(* Logix 5000 project; controller DispersionPlc vendor 1 type 14 code 108 rev 34.11; software revision 34.01; part 22 of 22 *)
(* tags used below, declared in another part *)
   AFI : BOOL;
   DeviationFactor : REAL;
   Estop : BOOL;
   Estop_Disp : ALIAS FOR Local:3:I.Data.1;
   FC_4302_1 : AStd_PIDInterface;
   FC_4302_1_AOI : AStd_PIDInterface_AOI;
   FC_4302_1_PID : PID_ENHANCED;
   FCV_4302_1 : AStd_VlvModulating;
   FIT_4302_2 : AStd_AnalogInput;
   GenPurp : AStd_GeneralPurp;
   LS_4302_High : BOOL;
   PLCStatus : AStd_PLCStatus;
   RO_HE4305_PhaseROWaterAddition : AStd_PLI;
   SV_4307_1 : AStd_VlvOC;
   TIT_4307_1 : AStd_AnalogInput;
   V4306_PhaseTransfer : AStd_PLI;
   V4307_PhaseCool : AStd_PLI;
   V4307_PhaseCool_AOI : AStd_PLI_AOI;
   V4307_PhaseRunPumpCirculate : AStd_PLI;
   V4307_PhaseRunPumpCirculate_AOI : AStd_PLI_AOI;
   V4307_PhaseTransfer : AStd_PLI;
   V4307_PhaseTransfer_AOI : AStd_PLI_AOI;
   V4307_PhaseTransfer_DelayTimer : TIMER;
   V4307_Transfer_LineClear : TIMER;
   VFD_4302_1 : AStd_VFD;
   VFD_4307_1 : AStd_VFD;
   WIT_4307_1 : AStd_AnalogInput;
   XV_4302_10 : AStd_VlvOC;
   XV_4306_5 : AStd_VlvOC;
   XV_4307_1 : AStd_VlvOC;
   XV_4307_2 : AStd_VlvOC;
   XV_4307_4 : AStd_VlvOC;
   XV_4307_6 : AStd_VlvOC;
(* Unit_V4307, continued *)

ROUTINE Phase_Cool   (* ladder *)
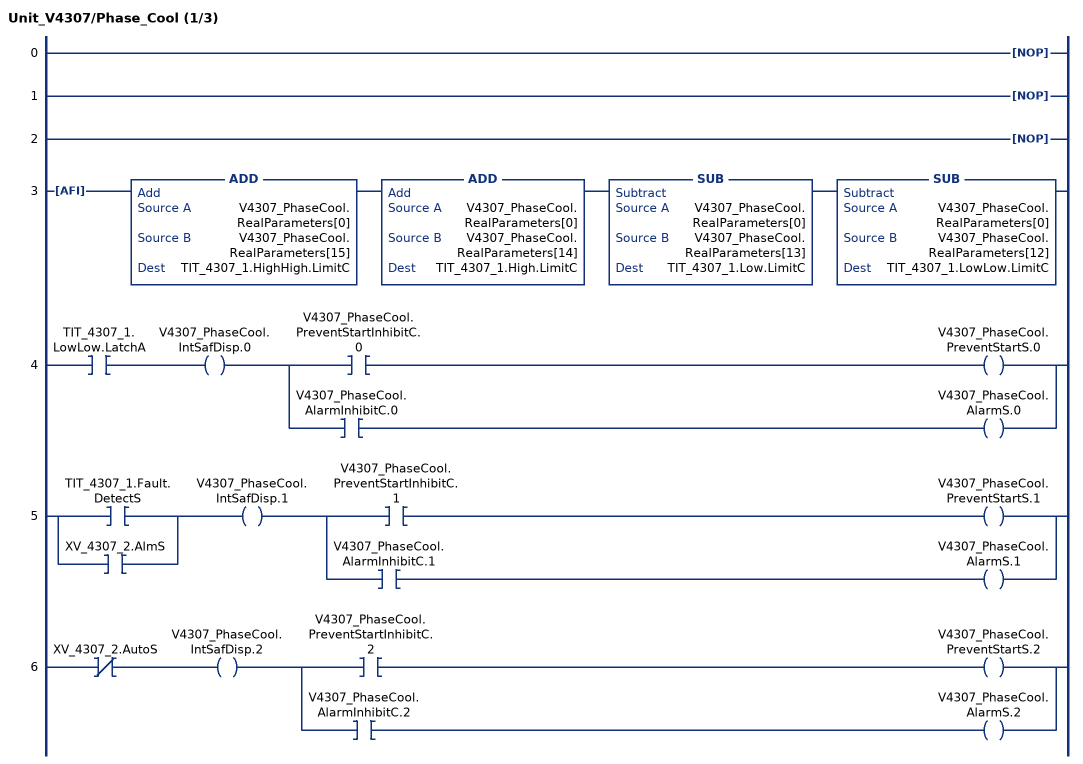
   0: NOP();
   1: NOP();
   2: NOP();
   3: AFI()ADD(V4307_PhaseCool.RealParameters[0],V4307_PhaseCool.RealParameters[15],TIT_4307_1.HighHigh.LimitC)ADD(V4307_PhaseCool.RealParameters[0],V4307_PhaseCool.RealParameters[14],TIT_4307_1.High.LimitC)SUB(V4307_PhaseCool.RealParameters[0],V4307_PhaseCool.RealParameters[13],TIT_4307_1.Low.LimitC)SUB(V4307_PhaseCool.RealParameters[0],V4307_PhaseCool.RealParameters[12],TIT_4307_1.LowLow.LimitC);
   4: XIC(TIT_4307_1.LowLow.LatchA)OTE(V4307_PhaseCool.IntSafDisp.0)[XIC(V4307_PhaseCool.PreventStartInhibitC.0) OTE(V4307_PhaseCool.PreventStartS.0) ,XIC(V4307_PhaseCool.AlarmInhibitC.0) OTE(V4307_PhaseCool.AlarmS.0) ];
   5: [XIC(TIT_4307_1.Fault.DetectS) ,XIC(XV_4307_2.AlmS) ]OTE(V4307_PhaseCool.IntSafDisp.1)[XIC(V4307_PhaseCool.PreventStartInhibitC.1) OTE(V4307_PhaseCool.PreventStartS.1) ,XIC(V4307_PhaseCool.AlarmInhibitC.1) OTE(V4307_PhaseCool.AlarmS.1) ];
   6: XIO(XV_4307_2.AutoS)OTE(V4307_PhaseCool.IntSafDisp.2)[XIC(V4307_PhaseCool.PreventStartInhibitC.2) OTE(V4307_PhaseCool.PreventStartS.2) ,XIC(V4307_PhaseCool.AlarmInhibitC.2) OTE(V4307_PhaseCool.AlarmS.2) ];
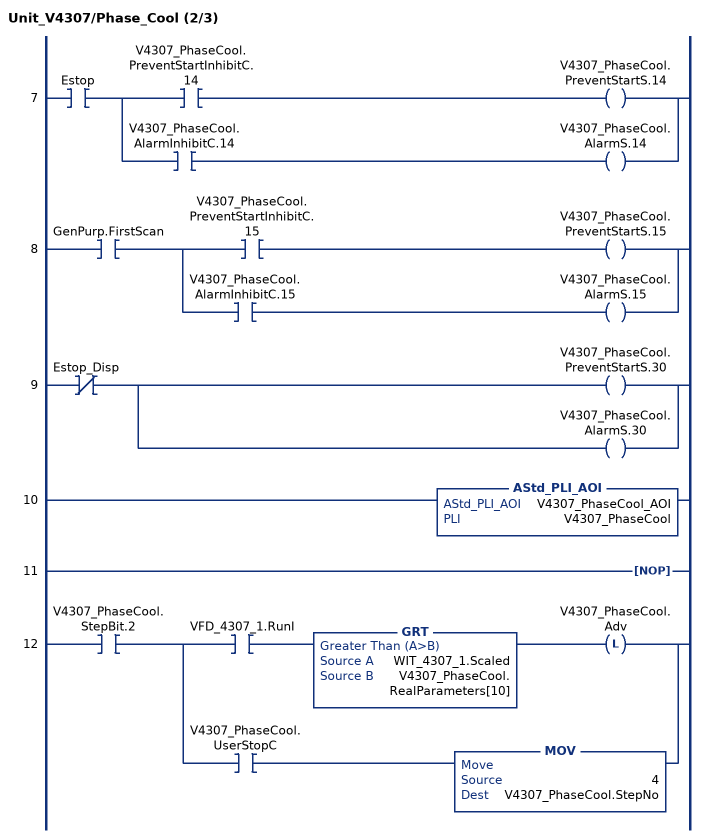
   7: XIC(Estop)[XIC(V4307_PhaseCool.PreventStartInhibitC.14) OTE(V4307_PhaseCool.PreventStartS.14) ,XIC(V4307_PhaseCool.AlarmInhibitC.14) OTE(V4307_PhaseCool.AlarmS.14) ];
   8: XIC(GenPurp.FirstScan)[XIC(V4307_PhaseCool.PreventStartInhibitC.15) OTE(V4307_PhaseCool.PreventStartS.15) ,XIC(V4307_PhaseCool.AlarmInhibitC.15) OTE(V4307_PhaseCool.AlarmS.15) ];
   9: XIO(Estop_Disp)[OTE(V4307_PhaseCool.PreventStartS.30) ,OTE(V4307_PhaseCool.AlarmS.30) ];
   10: AStd_PLI_AOI(V4307_PhaseCool_AOI,V4307_PhaseCool);
   11: NOP();
   12: XIC(V4307_PhaseCool.StepBit.2)[XIC(VFD_4307_1.RunI) GRT(WIT_4307_1.Scaled,V4307_PhaseCool.RealParameters[10]) OTL(V4307_PhaseCool.Adv) ,XIC(V4307_PhaseCool.UserStopC) MOV(4,V4307_PhaseCool.StepNo) ];
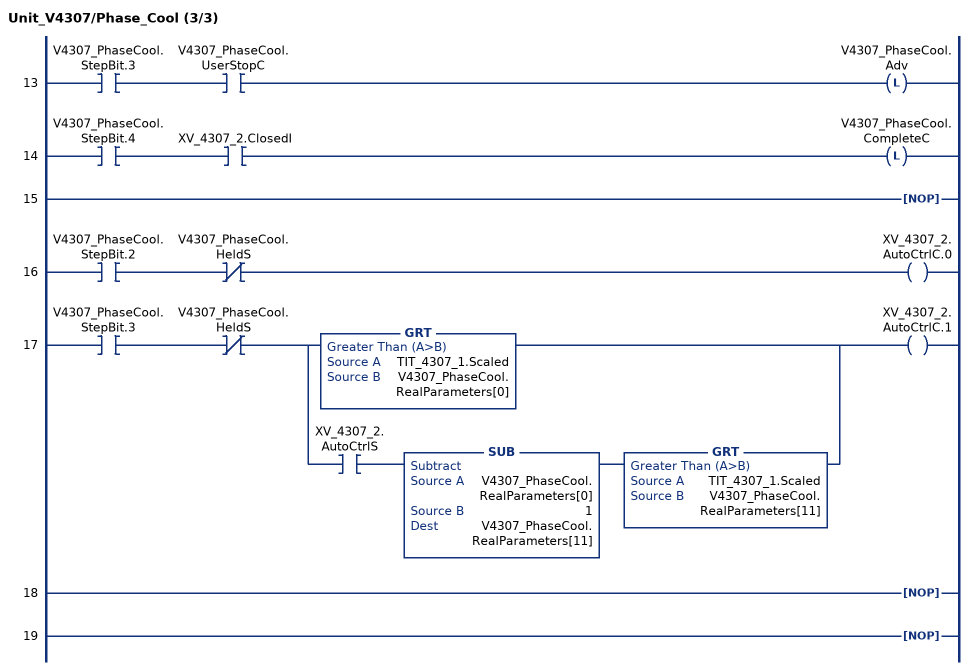
   13: XIC(V4307_PhaseCool.StepBit.3)XIC(V4307_PhaseCool.UserStopC)OTL(V4307_PhaseCool.Adv);
   14: XIC(V4307_PhaseCool.StepBit.4)XIC(XV_4307_2.ClosedI)OTL(V4307_PhaseCool.CompleteC);
   15: NOP();
   16: XIC(V4307_PhaseCool.StepBit.2)XIO(V4307_PhaseCool.HeldS)OTE(XV_4307_2.AutoCtrlC.0);
   17: XIC(V4307_PhaseCool.StepBit.3)XIO(V4307_PhaseCool.HeldS)[GRT(TIT_4307_1.Scaled,V4307_PhaseCool.RealParameters[0]) ,XIC(XV_4307_2.AutoCtrlS) SUB(V4307_PhaseCool.RealParameters[0],1,V4307_PhaseCool.RealParameters[11]) GRT(TIT_4307_1.Scaled,V4307_PhaseCool.RealParameters[11]) ]OTE(XV_4307_2.AutoCtrlC.1);
   18: NOP();
   19: NOP();
END_ROUTINE

ROUTINE Phase_RunPump_Circulate   (* ladder *)
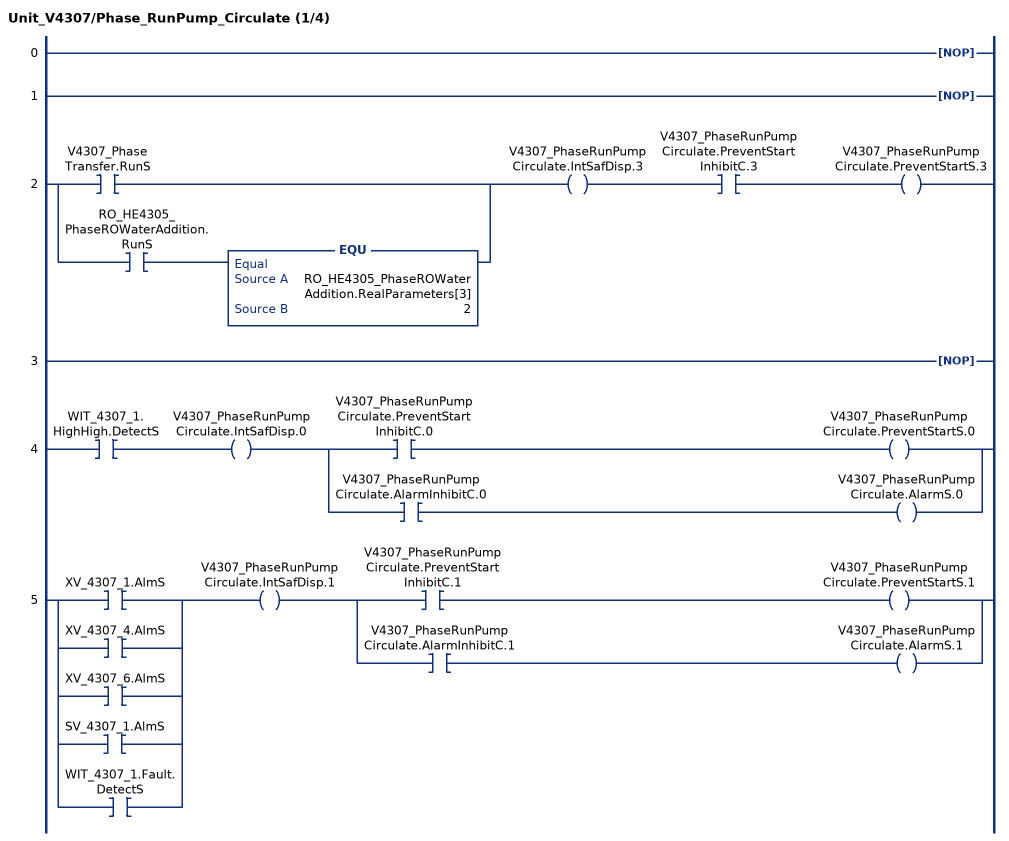
   0: NOP();
   1: NOP();
   2: [XIC(V4307_PhaseTransfer.RunS) ,XIC(RO_HE4305_PhaseROWaterAddition.RunS) EQU(RO_HE4305_PhaseROWaterAddition.RealParameters[3],2) ]OTE(V4307_PhaseRunPumpCirculate.IntSafDisp.3)XIC(V4307_PhaseRunPumpCirculate.PreventStartInhibitC.3)OTE(V4307_PhaseRunPumpCirculate.PreventStartS.3);
   3: NOP();
   4: XIC(WIT_4307_1.HighHigh.DetectS)OTE(V4307_PhaseRunPumpCirculate.IntSafDisp.0)[XIC(V4307_PhaseRunPumpCirculate.PreventStartInhibitC.0) OTE(V4307_PhaseRunPumpCirculate.PreventStartS.0) ,XIC(V4307_PhaseRunPumpCirculate.AlarmInhibitC.0) OTE(V4307_PhaseRunPumpCirculate.AlarmS.0) ];
   5: [XIC(XV_4307_1.AlmS) ,XIC(XV_4307_4.AlmS) ,XIC(XV_4307_6.AlmS) ,XIC(SV_4307_1.AlmS) ,XIC(WIT_4307_1.Fault.DetectS) ]OTE(V4307_PhaseRunPumpCirculate.IntSafDisp.1)[XIC(V4307_PhaseRunPumpCirculate.PreventStartInhibitC.1) OTE(V4307_PhaseRunPumpCirculate.PreventStartS.1) ,XIC(V4307_PhaseRunPumpCirculate.AlarmInhibitC.1) OTE(V4307_PhaseRunPumpCirculate.AlarmS.1) ];
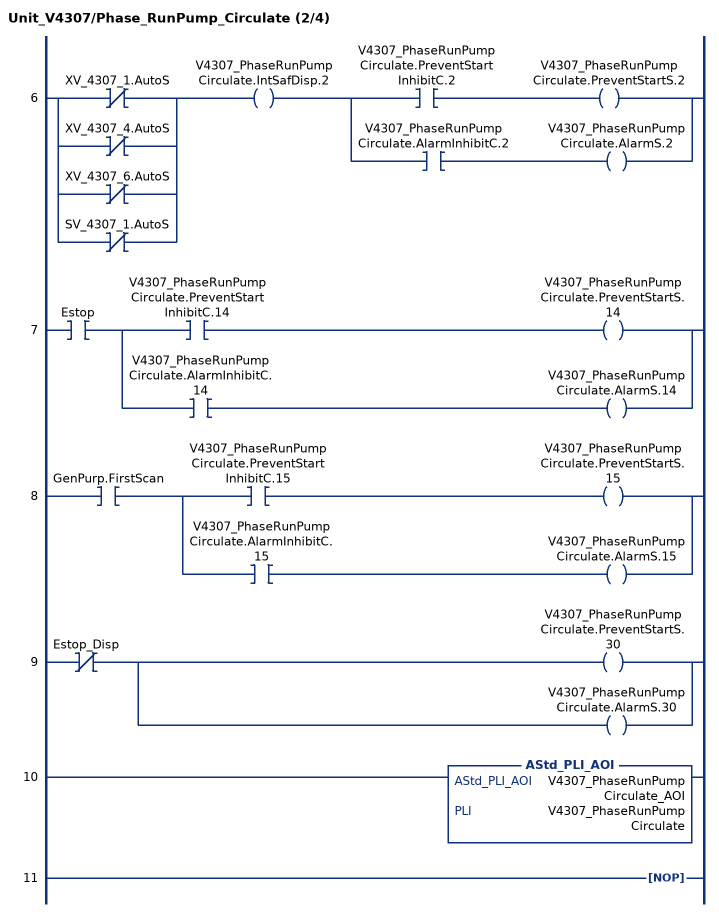
   6: [XIO(XV_4307_1.AutoS) ,XIO(XV_4307_4.AutoS) ,XIO(XV_4307_6.AutoS) ,XIO(SV_4307_1.AutoS) ]OTE(V4307_PhaseRunPumpCirculate.IntSafDisp.2)[XIC(V4307_PhaseRunPumpCirculate.PreventStartInhibitC.2) OTE(V4307_PhaseRunPumpCirculate.PreventStartS.2) ,XIC(V4307_PhaseRunPumpCirculate.AlarmInhibitC.2) OTE(V4307_PhaseRunPumpCirculate.AlarmS.2) ];
   7: XIC(Estop)[XIC(V4307_PhaseRunPumpCirculate.PreventStartInhibitC.14) OTE(V4307_PhaseRunPumpCirculate.PreventStartS.14) ,XIC(V4307_PhaseRunPumpCirculate.AlarmInhibitC.14) OTE(V4307_PhaseRunPumpCirculate.AlarmS.14) ];
   8: XIC(GenPurp.FirstScan)[XIC(V4307_PhaseRunPumpCirculate.PreventStartInhibitC.15) OTE(V4307_PhaseRunPumpCirculate.PreventStartS.15) ,XIC(V4307_PhaseRunPumpCirculate.AlarmInhibitC.15) OTE(V4307_PhaseRunPumpCirculate.AlarmS.15) ];
   9: XIO(Estop_Disp)[OTE(V4307_PhaseRunPumpCirculate.PreventStartS.30) ,OTE(V4307_PhaseRunPumpCirculate.AlarmS.30) ];
   10: AStd_PLI_AOI(V4307_PhaseRunPumpCirculate_AOI,V4307_PhaseRunPumpCirculate);
   11: NOP();
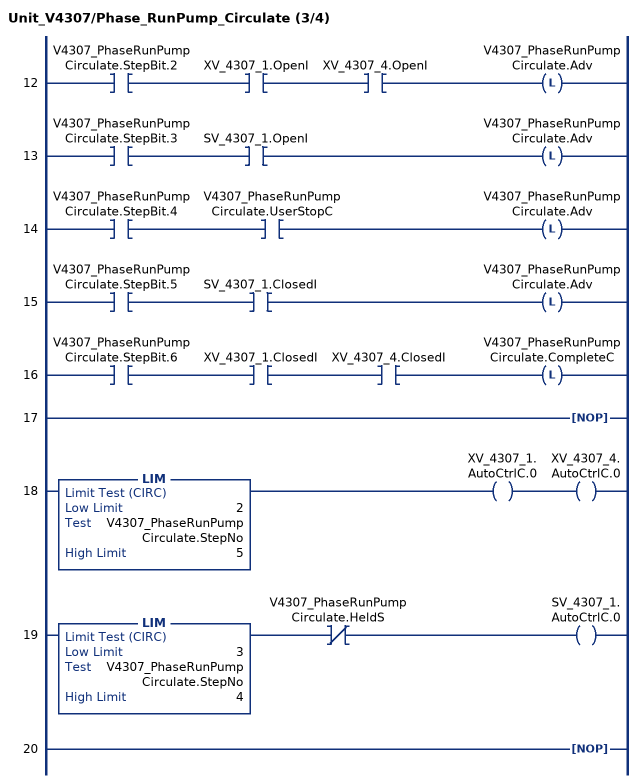
   12: XIC(V4307_PhaseRunPumpCirculate.StepBit.2)XIC(XV_4307_1.OpenI)XIC(XV_4307_4.OpenI)OTL(V4307_PhaseRunPumpCirculate.Adv);
   13: XIC(V4307_PhaseRunPumpCirculate.StepBit.3)XIC(SV_4307_1.OpenI)OTL(V4307_PhaseRunPumpCirculate.Adv);
   14: XIC(V4307_PhaseRunPumpCirculate.StepBit.4)XIC(V4307_PhaseRunPumpCirculate.UserStopC)OTL(V4307_PhaseRunPumpCirculate.Adv);
   15: XIC(V4307_PhaseRunPumpCirculate.StepBit.5)XIC(SV_4307_1.ClosedI)OTL(V4307_PhaseRunPumpCirculate.Adv);
   16: XIC(V4307_PhaseRunPumpCirculate.StepBit.6)XIC(XV_4307_1.ClosedI)XIC(XV_4307_4.ClosedI)OTL(V4307_PhaseRunPumpCirculate.CompleteC);
   17: NOP();
   18: LIM(2,V4307_PhaseRunPumpCirculate.StepNo,5)OTE(XV_4307_1.AutoCtrlC.0)OTE(XV_4307_4.AutoCtrlC.0);
   19: LIM(3,V4307_PhaseRunPumpCirculate.StepNo,4)XIO(V4307_PhaseRunPumpCirculate.HeldS)OTE(SV_4307_1.AutoCtrlC.0);
   20: NOP();
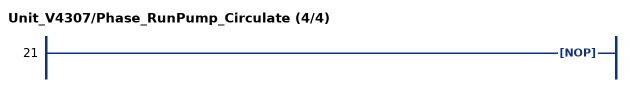
   21: NOP();
END_ROUTINE

ROUTINE Phase_Transfer   (* ladder *)
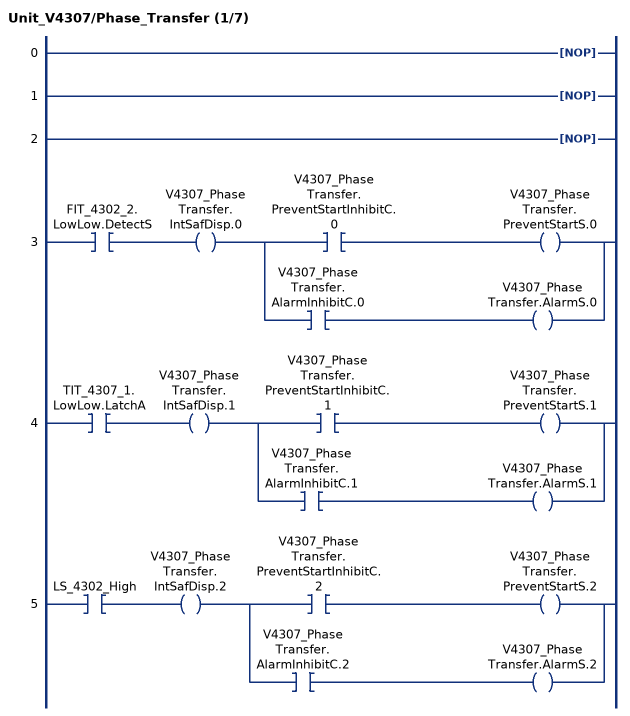
   0: NOP();
   1: NOP();
   2: NOP();
   3: XIC(FIT_4302_2.LowLow.DetectS)OTE(V4307_PhaseTransfer.IntSafDisp.0)[XIC(V4307_PhaseTransfer.PreventStartInhibitC.0) OTE(V4307_PhaseTransfer.PreventStartS.0) ,XIC(V4307_PhaseTransfer.AlarmInhibitC.0) OTE(V4307_PhaseTransfer.AlarmS.0) ];
   4: XIC(TIT_4307_1.LowLow.LatchA)OTE(V4307_PhaseTransfer.IntSafDisp.1)[XIC(V4307_PhaseTransfer.PreventStartInhibitC.1) OTE(V4307_PhaseTransfer.PreventStartS.1) ,XIC(V4307_PhaseTransfer.AlarmInhibitC.1) OTE(V4307_PhaseTransfer.AlarmS.1) ];
   5: XIC(LS_4302_High)OTE(V4307_PhaseTransfer.IntSafDisp.2)[XIC(V4307_PhaseTransfer.PreventStartInhibitC.2) OTE(V4307_PhaseTransfer.PreventStartS.2) ,XIC(V4307_PhaseTransfer.AlarmInhibitC.2) OTE(V4307_PhaseTransfer.AlarmS.2) ];
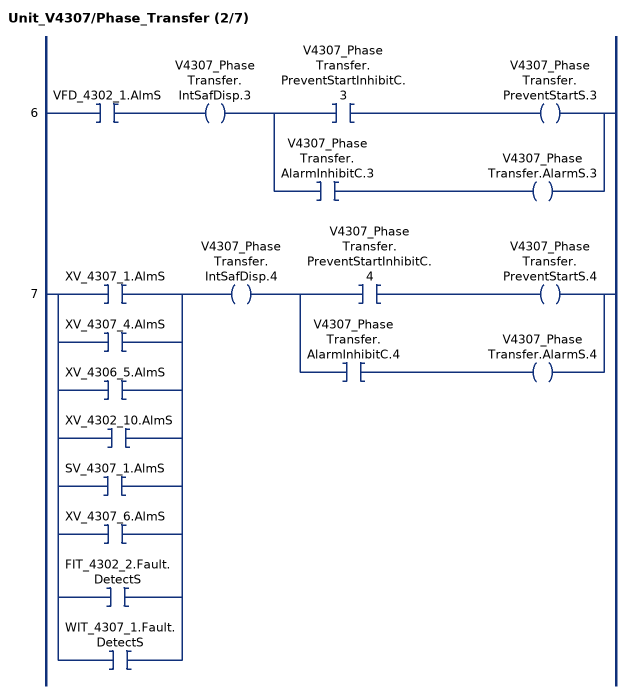
   6: XIC(VFD_4302_1.AlmS)OTE(V4307_PhaseTransfer.IntSafDisp.3)[XIC(V4307_PhaseTransfer.PreventStartInhibitC.3) OTE(V4307_PhaseTransfer.PreventStartS.3) ,XIC(V4307_PhaseTransfer.AlarmInhibitC.3) OTE(V4307_PhaseTransfer.AlarmS.3) ];
   7: [XIC(XV_4307_1.AlmS) ,XIC(XV_4307_4.AlmS) ,XIC(XV_4306_5.AlmS) ,XIC(XV_4302_10.AlmS) ,XIC(SV_4307_1.AlmS) ,XIC(XV_4307_6.AlmS) ,XIC(FIT_4302_2.Fault.DetectS) ,XIC(WIT_4307_1.Fault.DetectS) ]OTE(V4307_PhaseTransfer.IntSafDisp.4)[XIC(V4307_PhaseTransfer.PreventStartInhibitC.4) OTE(V4307_PhaseTransfer.PreventStartS.4) ,XIC(V4307_PhaseTransfer.AlarmInhibitC.4) OTE(V4307_PhaseTransfer.AlarmS.4) ];
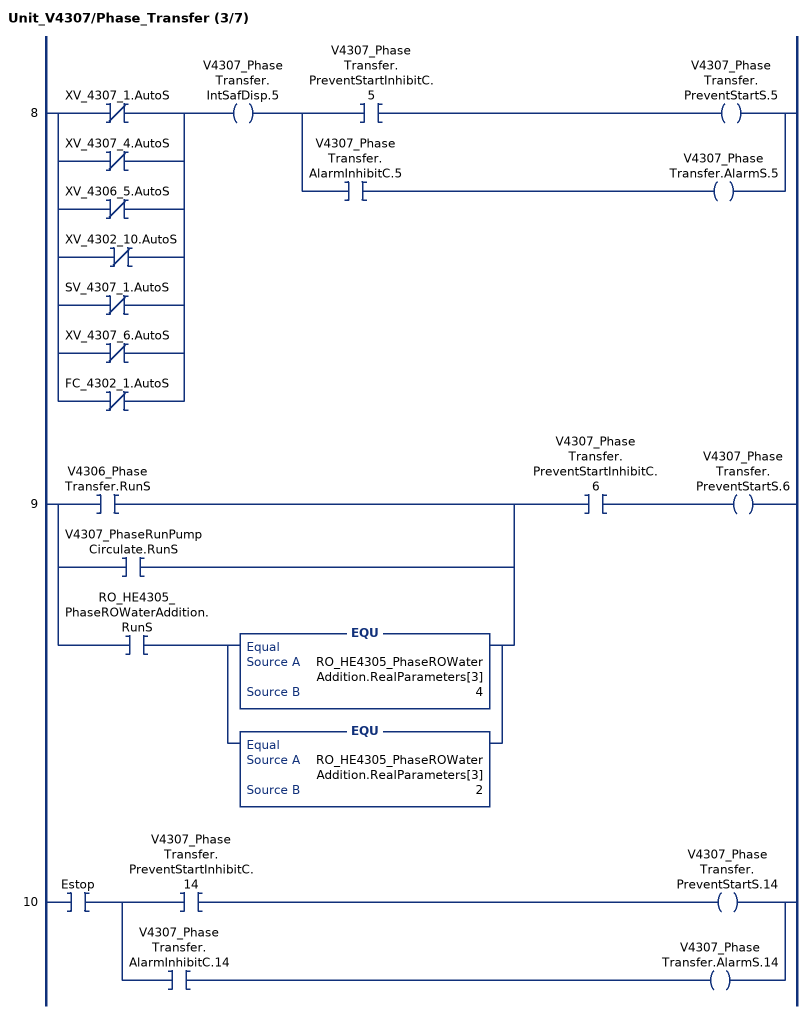
   8: [XIO(XV_4307_1.AutoS) ,XIO(XV_4307_4.AutoS) ,XIO(XV_4306_5.AutoS) ,XIO(XV_4302_10.AutoS) ,XIO(SV_4307_1.AutoS) ,XIO(XV_4307_6.AutoS) ,XIO(FC_4302_1.AutoS) ]OTE(V4307_PhaseTransfer.IntSafDisp.5)[XIC(V4307_PhaseTransfer.PreventStartInhibitC.5) OTE(V4307_PhaseTransfer.PreventStartS.5) ,XIC(V4307_PhaseTransfer.AlarmInhibitC.5) OTE(V4307_PhaseTransfer.AlarmS.5) ];
   9: [XIC(V4306_PhaseTransfer.RunS) ,XIC(V4307_PhaseRunPumpCirculate.RunS) ,XIC(RO_HE4305_PhaseROWaterAddition.RunS) [EQU(RO_HE4305_PhaseROWaterAddition.RealParameters[3],4) ,EQU(RO_HE4305_PhaseROWaterAddition.RealParameters[3],2) ] ]XIC(V4307_PhaseTransfer.PreventStartInhibitC.6)OTE(V4307_PhaseTransfer.PreventStartS.6);
   10: XIC(Estop)[XIC(V4307_PhaseTransfer.PreventStartInhibitC.14) OTE(V4307_PhaseTransfer.PreventStartS.14) ,XIC(V4307_PhaseTransfer.AlarmInhibitC.14) OTE(V4307_PhaseTransfer.AlarmS.14) ];
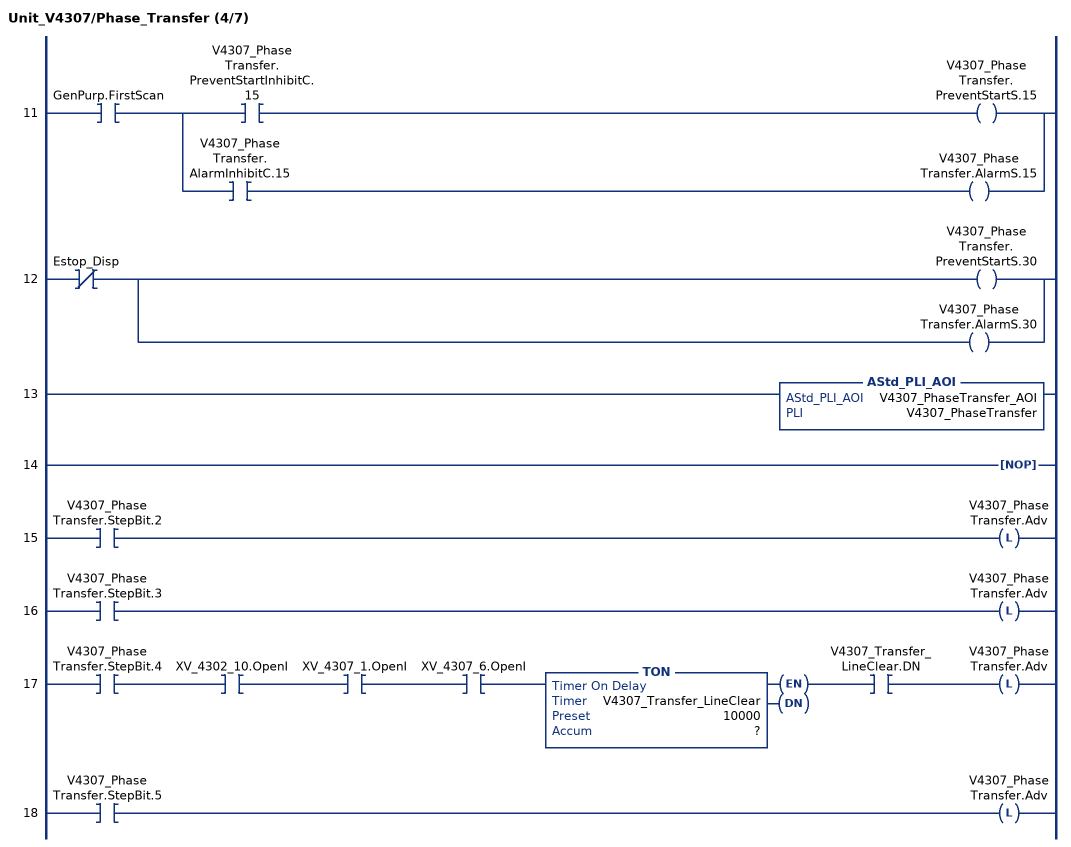
   11: XIC(GenPurp.FirstScan)[XIC(V4307_PhaseTransfer.PreventStartInhibitC.15) OTE(V4307_PhaseTransfer.PreventStartS.15) ,XIC(V4307_PhaseTransfer.AlarmInhibitC.15) OTE(V4307_PhaseTransfer.AlarmS.15) ];
   12: XIO(Estop_Disp)[OTE(V4307_PhaseTransfer.PreventStartS.30) ,OTE(V4307_PhaseTransfer.AlarmS.30) ];
   13: AStd_PLI_AOI(V4307_PhaseTransfer_AOI,V4307_PhaseTransfer);
   14: NOP();
   15: XIC(V4307_PhaseTransfer.StepBit.2)OTL(V4307_PhaseTransfer.Adv);
   16: XIC(V4307_PhaseTransfer.StepBit.3)OTL(V4307_PhaseTransfer.Adv);
   17: XIC(V4307_PhaseTransfer.StepBit.4)XIC(XV_4302_10.OpenI)XIC(XV_4307_1.OpenI)XIC(XV_4307_6.OpenI)TON(V4307_Transfer_LineClear,?,?)XIC(V4307_Transfer_LineClear.DN)OTL(V4307_PhaseTransfer.Adv);
   18: XIC(V4307_PhaseTransfer.StepBit.5)OTL(V4307_PhaseTransfer.Adv);
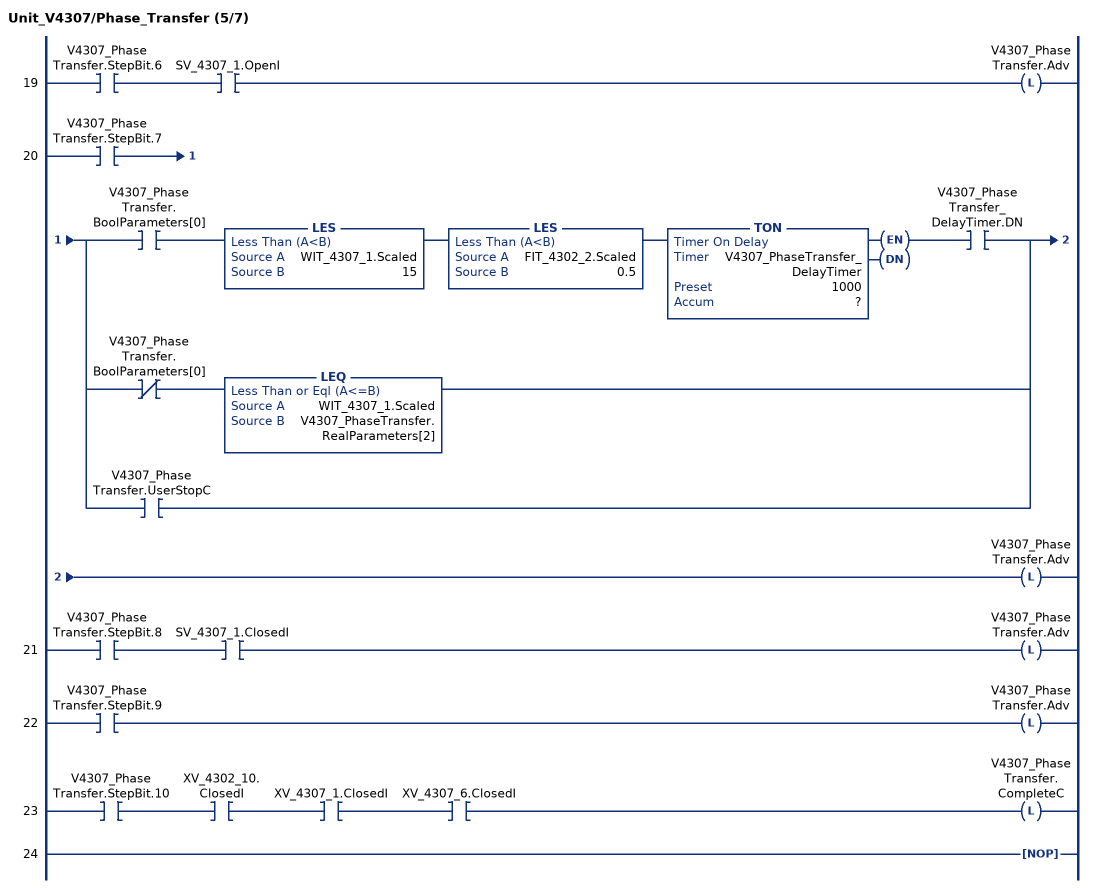
   19: XIC(V4307_PhaseTransfer.StepBit.6)XIC(SV_4307_1.OpenI)OTL(V4307_PhaseTransfer.Adv);
   20: XIC(V4307_PhaseTransfer.StepBit.7)[XIC(V4307_PhaseTransfer.BoolParameters[0]) LES(WIT_4307_1.Scaled,15) LES(FIT_4302_2.Scaled,0.5) TON(V4307_PhaseTransfer_DelayTimer,?,?) XIC(V4307_PhaseTransfer_DelayTimer.DN) ,XIO(V4307_PhaseTransfer.BoolParameters[0]) LEQ(WIT_4307_1.Scaled,V4307_PhaseTransfer.RealParameters[2]) ,XIC(V4307_PhaseTransfer.UserStopC) ]OTL(V4307_PhaseTransfer.Adv);
   21: XIC(V4307_PhaseTransfer.StepBit.8)XIC(SV_4307_1.ClosedI)OTL(V4307_PhaseTransfer.Adv);
   22: XIC(V4307_PhaseTransfer.StepBit.9)OTL(V4307_PhaseTransfer.Adv);
   23: XIC(V4307_PhaseTransfer.StepBit.10)XIC(XV_4302_10.ClosedI)XIC(XV_4307_1.ClosedI)XIC(XV_4307_6.ClosedI)OTL(V4307_PhaseTransfer.CompleteC);
   24: NOP();
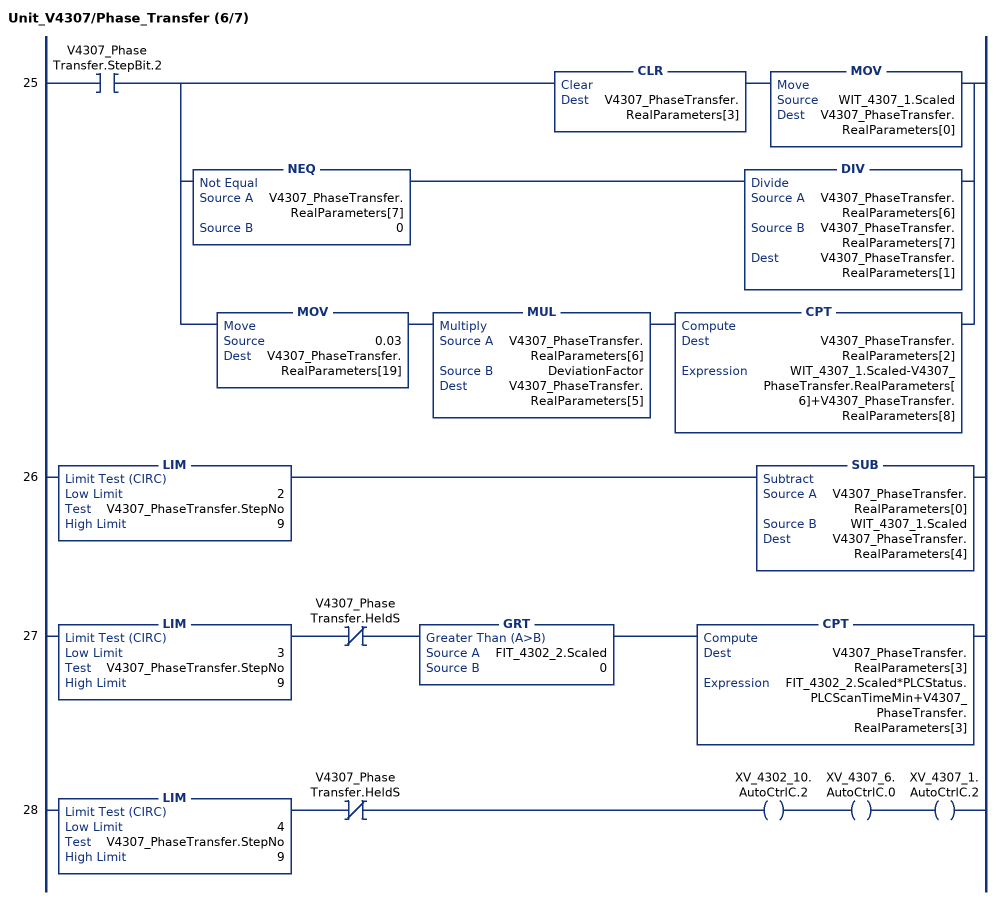
   25: XIC(V4307_PhaseTransfer.StepBit.2)[CLR(V4307_PhaseTransfer.RealParameters[3]) MOV(WIT_4307_1.Scaled,V4307_PhaseTransfer.RealParameters[0]) ,NEQ(V4307_PhaseTransfer.RealParameters[7],0) DIV(V4307_PhaseTransfer.RealParameters[6],V4307_PhaseTransfer.RealParameters[7],V4307_PhaseTransfer.RealParameters[1]) ,MOV(0.03,V4307_PhaseTransfer.RealParameters[19]) MUL(V4307_PhaseTransfer.RealParameters[6],DeviationFactor,V4307_PhaseTransfer.RealParameters[5]) CPT(V4307_PhaseTransfer.RealParameters[2],WIT_4307_1.Scaled-V4307_PhaseTransfer.RealParameters[6]+V4307_PhaseTransfer.RealParameters[8]) ];
   26: LIM(2,V4307_PhaseTransfer.StepNo,9)SUB(V4307_PhaseTransfer.RealParameters[0],WIT_4307_1.Scaled,V4307_PhaseTransfer.RealParameters[4]);
   27: LIM(3,V4307_PhaseTransfer.StepNo,9)XIO(V4307_PhaseTransfer.HeldS)GRT(FIT_4302_2.Scaled,0)CPT(V4307_PhaseTransfer.RealParameters[3],FIT_4302_2.Scaled*PLCStatus.PLCScanTimeMin+V4307_PhaseTransfer.RealParameters[3]);
   28: LIM(4,V4307_PhaseTransfer.StepNo,9)XIO(V4307_PhaseTransfer.HeldS)OTE(XV_4302_10.AutoCtrlC.2)OTE(XV_4307_6.AutoCtrlC.0)OTE(XV_4307_1.AutoCtrlC.2);
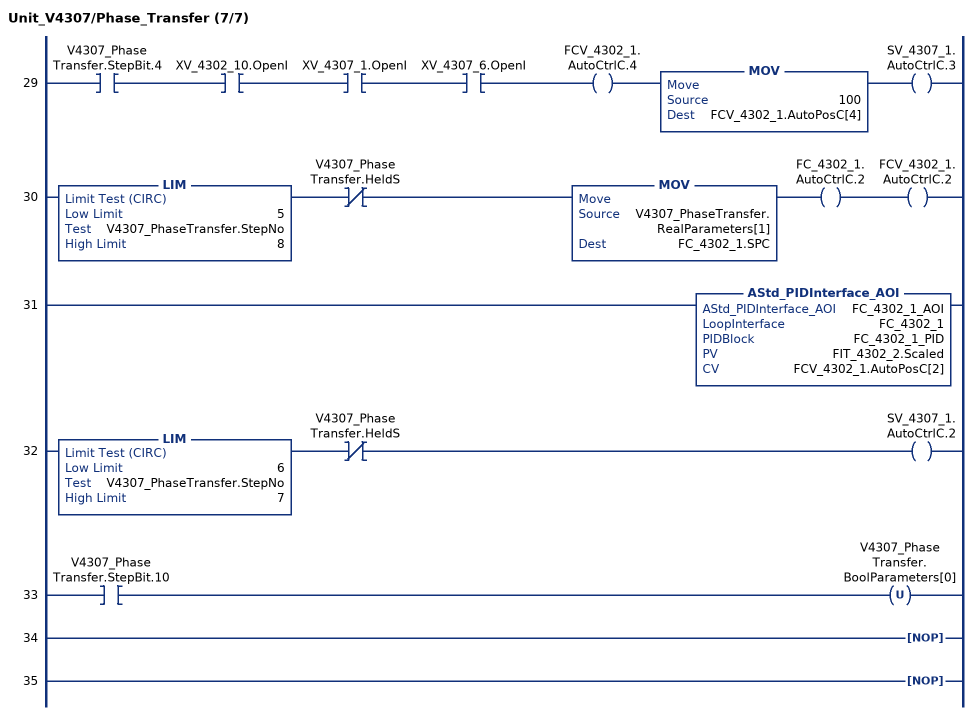
   29: XIC(V4307_PhaseTransfer.StepBit.4)XIC(XV_4302_10.OpenI)XIC(XV_4307_1.OpenI)XIC(XV_4307_6.OpenI)OTE(FCV_4302_1.AutoCtrlC.4)MOV(100,FCV_4302_1.AutoPosC[4])OTE(SV_4307_1.AutoCtrlC.3);
   30: LIM(5,V4307_PhaseTransfer.StepNo,8)XIO(V4307_PhaseTransfer.HeldS)MOV(V4307_PhaseTransfer.RealParameters[1],FC_4302_1.SPC)OTE(FC_4302_1.AutoCtrlC.2)OTE(FCV_4302_1.AutoCtrlC.2);
   31: AStd_PIDInterface_AOI(FC_4302_1_AOI,FC_4302_1,FC_4302_1_PID,FIT_4302_2.Scaled,FCV_4302_1.AutoPosC[2]);
   32: LIM(6,V4307_PhaseTransfer.StepNo,7)XIO(V4307_PhaseTransfer.HeldS)OTE(SV_4307_1.AutoCtrlC.2);
   33: XIC(V4307_PhaseTransfer.StepBit.10)OTU(V4307_PhaseTransfer.BoolParameters[0]);
   34: NOP();
   35: NOP();
END_ROUTINE
END_PROGRAM
